TYPE E_DataExchaSteps :
(
	DATAEXCHA_STATE_IDLE,
	DATAEXCHA_STATE_SEND_START,
	DATAEXCHA_STATE_SEND_WAIT,
	DATAEXCHA_STATE_RECEIVE_START,
	DATAEXCHA_STATE_RECEIVE_WAIT,
	DATAEXCHA_STATE_ERROR,
	DATAEXCHA_STATE_RECEIVE_BEFORE_RETRY_START,
	DATAEXCHA_STATE_RECEIVE_BEFORE_RETRY_WAIT
);
END_TYPE

(* stored: Version 1.1.0.1, ProductVersion 3.1.4024.10
   DUT E_DataExchaSteps: Id {cb9b548c-a5a2-4d36-9ee1-a99a9f31a932} *)
